FUNCTION_BLOCK FB_ReceiveVelocityIntegral_Right
VAR_IN_OUT
	Inputs_Right : CANRXQUEUESTRUCT_E_32;
	Outputs_Right : CANTXQUEUESTRUCT_E_32;
END_VAR
VAR_OUTPUT
	VelocityIntegral_Right : LREAL;
END_VAR
VAR
	MessageReceived : ARRAY[0..31] OF EXTCANQUEUE;
	i : INT;
	
	fbPPS_Timer : TON;
	nPacketsPerSecond: INT;
	nReceiveCounter : INT;
	nLastReceiveCounter : INT;
END_VAR

FOR i := 0 TO (Inputs_Right.NoOfRxMessages-1) DO
    IF Inputs_Right.RxMessages[i].cobId = 1500 THEN 
       VelocityIntegral_Right := INT_TO_LREAL(DWORD_TO_INT(SHL(USINT_TO_UDINT(Inputs_Right.RxMessages[i].data[0]), 24) OR SHL(USINT_TO_UDINT(Inputs_Right.RxMessages[i].data[1]), 16) OR SHL(USINT_TO_UDINT(Inputs_Right.RxMessages[i].data[2]), 8)  OR USINT_TO_UDINT(Inputs_Right.RxMessages[i].data[3]))) / 100.0; 
         
    	nReceiveCounter := nReceiveCounter + 1;
	END_IF
END_FOR
fbPPS_Timer(IN := NOT fbPPS_Timer.Q, PT := T#1S);
IF fbPPS_Timer.Q THEN
			nPacketsPerSecond   := nReceiveCounter - nLastReceiveCounter;
			nLastReceiveCounter := nReceiveCounter;
END_IF

END_FUNCTION_BLOCK

(* stored: Version 1.1.0.1
   POU FB_ReceiveVelocityIntegral_Right: Id {de2f069d-fa57-4de1-8d68-b4a91e77c6d0}, SpecialFunc None *)
